{attribute 'qualified_only'}
{attribute 'strict'}
{attribute 'to_string'}
TYPE E_Cylinder :
(
    Jib   := 1,
    Main  := 2
);
END_TYPE

(* stored: Version 1.1.0.1
   DUT E_Cylinder: Id {4c3e23a9-3b11-40ad-8d17-b0c7060e57c6} *)
